# EPICS autosave request: specsAnalyserApp/Db/specsAnalyser.req
$(P)$(R)DATA_DELAY_MAX
$(P)$(R)SAMPLES
$(P)$(R)VALUES
$(P)$(R)SLICES
$(P)$(R)LENS_MODE
$(P)$(R)SCAN_RANGE
$(P)$(R)ACQ_MODE
$(P)$(R)PASS_ENERGY
$(P)$(R)LOW_ENERGY
$(P)$(R)HIGH_ENERGY
$(P)$(R)KINETIC_ENERGY
$(P)$(R)RETARDING_RATIO
$(P)$(R)STEP_SIZE
